(* PLC project Generated.project, CODESYS CODESYS V3.5 SP19 Patch 1 *)
(* stored: creationDateTime 2026-09-06T13:00:42.579718, modificationDateTime 2026-09-06T13:00:42.579718 *)

{attribute 'qualified_only'}
VAR_GLOBAL  (* GVL_Global - ═══════════════════════════════════════════════════════════════ 🌐 GVL_Global — Variables globales d'utilité générale ─────────────────────────────────────────────────────────────── 🎯 Rôle : Horloges et signaux système partagés non persistants. 📄 Docs : DOC/AF/AF_Partie-02_Architecture_Programme_v3.2.md ═══════════════════════════════════════════════════════════════ *)
  BlinkClock : BOOL;  (* Horloge clignotement système (IHM/diag), rythme réglable GVL_PERSISTENT *)
END_VAR
